Staubli VAL3: onBackSpace.pgx

program onBackSpace(tool& x_tTool[])
begin
  //
  // NB sEvent is the selected
  // element in the LIST
  //
  if nIndex==0
    call editTool(x_tTool.trsf)
    call tcp:setTool(x_tTool,nIndexTool)
    logMsg("[VALlaser] INTERFACE:Change value of the tool :"+toString("",nIndexTool))
  endIf
  //
end
